TYPE ST_HMI_MANUAL_DRIVE_IN :
STRUCT
	eJogMode		: E_Drive_JogMode;
	stButtonJogPos,
	stButtonJogNeg,
	stButtonStop	: ST_HMI_BUTTON_IN;
END_STRUCT
END_TYPE

(* stored: Version 1.1.0.1, ProductVersion 3.1.4024.12
   DUT ST_HMI_MANUAL_DRIVE_IN: Id {3538a068-d5d2-4db9-84bf-1bffe3b8365c} *)
